FUNCTION_BLOCK AUI_TO_AUI2 (* Composite FB for convert unidirectional AUI to bidirectional AUI2 *)
  (* Standard: 61499-2; Function: AUI_IN publishes its value onto the outgoing (EO1) side of AUI2_BIDIR. Whatever AUI2_BIDIR receives on its incoming (EI1) side is forwarded out again as a plain unidirectional signal via AUI_OUT.; Description: Copyright (c) 2026 HR Agrartechnik GmbH This program and the accompanying materials are made available under the terms of the Eclipse Public License 2.0 which is available at https://www.eclipse.org/legal/epl-2.0/ SPDX-License-Identifier: EPL-2.0 *)
  (* Version 1.0, 2026-09-12, Franz Höpfinger, HR Agrartechnik GmbH, Initial Version - Konvertierungsfamilie vervollstaendigt (analog zu AR2/AB2/AE2). *)
  PACKAGE adapter::conversion::bidirectional;
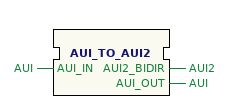
  SOCKETS
    AUI_IN : adapter::types::unidirectional::AUI; (* Adapter Input: unidirectional source *)
  END_SOCKETS
  PLUGS
    AUI2_BIDIR : adapter::types::bidirectional::AUI2; (* Adapter Output: bidirectional tap, outgoing side driven by AUI_IN, incoming side forwarded to AUI_OUT *)
    AUI_OUT : adapter::types::unidirectional::AUI; (* Adapter Output: mirrors AUI2_BIDIR's incoming (request) side *)
  END_PLUGS
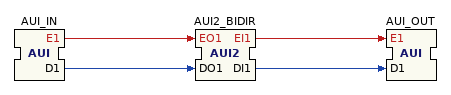
  EVENT_CONNECTIONS
    AUI_IN.E1 TO AUI2_BIDIR.EO1;
    AUI2_BIDIR.EI1 TO AUI_OUT.E1;
  END_CONNECTIONS
  DATA_CONNECTIONS
    AUI_IN.D1 TO AUI2_BIDIR.DO1;
    AUI2_BIDIR.DI1 TO AUI_OUT.D1;
  END_CONNECTIONS
END_FUNCTION_BLOCK
